// TwinCAT 3 PLC project RobotPlc
// ProgramVersion: 3.1.4024.0
// libraries:
//   Tc2_Standard, * (Beckhoff Automation GmbH)
//   Tc2_System, * (Beckhoff Automation GmbH)
//   Tc3_Module, * (Beckhoff Automation GmbH)
// project tree:
//   DUTs/ ST_FRUOPIn.TcDUT, ST_FRUOPOut.TcDUT, ST_FRConnection.TcDUT
//   / PlcTask.TcTTO
//   POUs/ FB_FRPower.TcPOU, FB_FRProgSelect.TcPOU, MAIN.TcPOU
// real-time tasks:
//   TASK PlcTask: cycle T#10ms, priority 20, ADS port 350
//   TASK EIP Scanner Task: cycle T#1ms, priority 1, ADS port 301
// I/O:
//   DEVICE Device 1 (TC3 EIP Scanner), AmsNetId 192.168.100.3.2.1
//     FANUC Robot R30iB+ // <INFO> 192.168.2.2, FANUC Robot R30iB+ (ProdCode: 4, Rev: 3.01, Mac: 8c:8c:aa:d6:16:77) </INFO> <EDS> C:\TwinCAT\3.1\Config\Io\EtherNetIP\FANUCROBOT_EIP_V900.EDS </EDS>
// variable links:
//   RobotPlc/RobotPlc Instance <-> Device 1 (TC3 EIP Scanner)/FANUC Robot R30iB+
//     PlcTask Inputs/MAIN.stFRConnection._EIPConnectionState <-> Inputs/State
//     PlcTask Inputs/MAIN.stFRConnection._rawIn <-> Connection 1 (Input/Output)/Inputs/noname0_arrBYTE[0]
//     PlcTask Inputs/MAIN.stFRConnection._rawIn @bit {8..56 step 8} <-> Connection 1 (Input/Output)/Inputs/noname0_arrBYTE[{1..7}]  (7 links)
//     PlcTask Outputs/MAIN.stFRConnection._rawOut <-> Connection 1 (Input/Output)/Outputs/noname0_arrBYTE[0]
//     PlcTask Outputs/MAIN.stFRConnection._rawOut @bit {8..56 step 8} <-> Connection 1 (Input/Output)/Outputs/noname0_arrBYTE[{1..7}]  (7 links)

CONFIGURATION RobotPlc
    RESOURCE PLC ON TwinCAT3
        TASK PlcTask(INTERVAL := T#10ms, PRIORITY := 20);
        PROGRAM MAIN WITH PlcTask : MAIN;
    END_RESOURCE
END_CONFIGURATION

// ---- DUTs/ST_FRUOPIn.TcDUT
TYPE ST_FRUOPIn :
STRUCT
	UI01_IMSTP : BIT;
	UI02_Hold : BIT;
	UI03_SFSPD : BIT;
	UI04_CycleStop : BIT;
	UI05_FaultReset : BIT;
	UI06_Start : BIT;
	UI07_Home : BIT;
	UI08_Enable : BIT;
	UI09_RSR1_PNS1 : BIT;
	UI10_RSR2_PNS2 : BIT;
	UI11_RSR3_PNS3 : BIT;
	UI12_RSR4_PNS4 : BIT;
	UI13_RSR5_PNS5 : BIT;
	UI14_RSR6_PNS6 : BIT;
	UI15_RSR7_PNS7 : BIT;
	UI16_RSR8_PNS8 : BIT;
	UI17_PNSStrobe : BIT;
	UI18_ProdStart : BIT;
	UI19,UI20,UI21,UI22
	,UI23,UI24,UI25,UI26
	,UI27,UI28,UI29,UI30
	,UI31,UI32 : BIT;
END_STRUCT
END_TYPE

// ---- DUTs/ST_FRUOPOut.TcDUT
TYPE ST_FRUOPOut :
STRUCT
	UO01_CmdEnabled : BIT;
	UO02_SystemReady : BIT;
	UO03_PrgRunning : BIT;
	UO04_PrgPaused : BIT;
	UO05_MotionHeld : BIT;
	UO06_Fault : BIT;
	UO07_AtPerch : BIT;
	UO08_TPEnabled : BIT;
	UO09_BattAlarm : BIT;
	UO10_Busy : BIT;
	UO11_ACK1_SNO1 : BIT;
	UO12_ACK2_SNO2 : BIT;
	UO13_ACK3_SNO3 : BIT;
	UO14_ACK4_SNO4 : BIT;
	UO15_ACK5_SNO5 : BIT;
	UO16_ACK6_SNO6 : BIT;
	UO17_ACK7_SNO7 : BIT;
	UO18_ACK8_SNO8 : BIT;
	UO19_SNACK : BIT;
	UO20_Reserved : BIT;
	UO21,UO22,UO23
	,UO24,UO25,UO26
	,UO27,UO28,UO29
	,UO30,UO31,UO32 : BIT;
END_STRUCT
END_TYPE

// ---- DUTs/ST_FRConnection.TcDUT
TYPE ST_FRConnection :
STRUCT
	_EIPConnectionState AT %I* : UINT;
	_rawIn AT %I*:ARRAY[0..7] OF BYTE;
	_rawOut AT %Q*:ARRAY[0..7] OF BYTE;
END_STRUCT
END_TYPE

// ---- POUs/MAIN.TcPOU
PROGRAM MAIN
VAR
	stFRConnection : ST_FRConnection;
	fbFRPower : FB_FRPower;
	fbFRProgSelect : FB_FRProgSelect;
	
	bIMSTP : BOOL;
	bHold : BOOL;
	bSFSPD : BOOL;
	bCycleStop : BOOL;
	bFaultReset : BOOL;
	bStart : BOOL;
	bHome : BOOL;
	bEnable : BOOL;

	bCmdEnabled : BOOL;
	bSystemReady : BOOL;
	bPrgRunning : BOOL;
	bPrgPaused : BOOL;
	bMotionHeld : BOOL;
	bFault : BOOL;
	bAtPerch : BOOL;
	bTPEnabled : BOOL;
	bBattAlarm : BOOL;
	bBusy : BOOL;
	
	bProgSelectExec : BOOL;
	bProgSelectDone : BOOL;
	bProgSelectBusy : BOOL;
	nProgSelectNo : USINT;
	nSelectedProgNo : USINT;
END_VAR

FRTest();

ACTION FRTest:
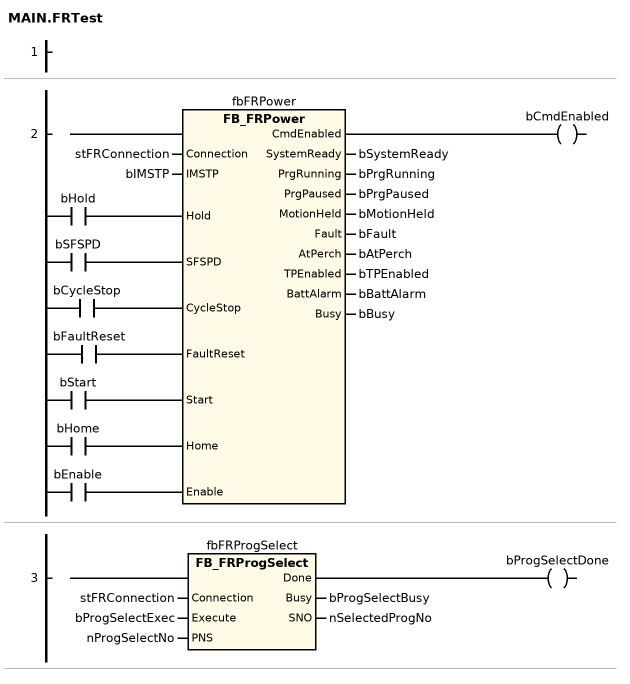
// NETWORK 1

// NETWORK 2
fbFRPower(
    Connection := stFRConnection,
    IMSTP := bIMSTP,
    Hold := bHold,
    SFSPD := bSFSPD,
    CycleStop := bCycleStop,
    FaultReset := bFaultReset,
    Start := bStart,
    Home := bHome,
    Enable := bEnable,
    SystemReady => bSystemReady,
    PrgRunning => bPrgRunning,
    PrgPaused => bPrgPaused,
    MotionHeld => bMotionHeld,
    Fault => bFault,
    AtPerch => bAtPerch,
    TPEnabled => bTPEnabled,
    BattAlarm => bBattAlarm,
    Busy => bBusy); // FB_FRPower
bCmdEnabled := fbFRPower.CmdEnabled;

// NETWORK 3
fbFRProgSelect(
    Connection := stFRConnection,
    Execute := bProgSelectExec,
    PNS := nProgSelectNo,
    Busy => bProgSelectBusy,
    SNO => nSelectedProgNo); // FB_FRProgSelect
bProgSelectDone := fbFRProgSelect.Done;
END_ACTION

END_PROGRAM

// ---- POUs/FB_FRPower.TcPOU
FUNCTION_BLOCK FB_FRPower
VAR_INPUT
	Connection : REFERENCE TO ST_FRConnection;
	IMSTP : BOOL;
	Hold : BOOL;
	SFSPD : BOOL;
	CycleStop : BOOL;
	FaultReset : BOOL;
	Start : BOOL;
	Home : BOOL;
	Enable : BOOL;
END_VAR
VAR_OUTPUT
	CmdEnabled : BOOL;
	SystemReady : BOOL;
	PrgRunning : BOOL;
	PrgPaused : BOOL;
	MotionHeld : BOOL;
	Fault : BOOL;
	AtPerch : BOOL;
	TPEnabled : BOOL;
	BattAlarm : BOOL;
	Busy : BOOL;
END_VAR
VAR
	stFRUOPIn : POINTER TO ST_FRUOPIn;
	stFRUOPOut : POINTER TO ST_FRUOPOut;
END_VAR

stFRUOPIn := ADR(Connection._rawOut);
stFRUOPOut := ADR(Connection._rawIn);

stFRUOPIn^.UI01_IMSTP := IMSTP;
stFRUOPIn^.UI02_Hold := Hold;
stFRUOPIn^.UI03_SFSPD := SFSPD;
stFRUOPIn^.UI04_CycleStop := CycleStop;
stFRUOPIn^.UI05_FaultReset := FaultReset;
stFRUOPIn^.UI06_Start := Start;
stFRUOPIn^.UI07_Home := Home;
stFRUOPIn^.UI08_Enable := Enable;

CmdEnabled := stFRUOPOut^.UO01_CmdEnabled;
SystemReady := stFRUOPOut^.UO02_SystemReady;
PrgRunning := stFRUOPOut^.UO03_PrgRunning;
PrgPaused := stFRUOPOut^.UO04_PrgPaused;
MotionHeld := stFRUOPOut^.UO05_MotionHeld;
Fault := stFRUOPOut^.UO06_Fault;
AtPerch := stFRUOPOut^.UO07_AtPerch;
TPEnabled := stFRUOPOut^.UO08_TPEnabled;
BattAlarm := stFRUOPOut^.UO09_BattAlarm;
Busy := stFRUOPOut^.UO09_BattAlarm;

END_FUNCTION_BLOCK

// ---- POUs/FB_FRProgSelect.TcPOU
FUNCTION_BLOCK FB_FRProgSelect
VAR_INPUT
	Connection : REFERENCE TO ST_FRConnection;
	Execute : BOOL;
	PNS : USINT;
END_VAR
VAR_OUTPUT
	Done : BOOL;
	Busy : BOOL;
	SNO : USINT;
END_VAR
VAR
	stFRUOPIn : POINTER TO ST_FRUOPIn;
	stFRUOPOut : POINTER TO ST_FRUOPOut;
	
	eProgState : (WAIT_EXEC, PNSSTROBE_TRIG, PNSSTROBE, WAIT_SNACK_DOWN, PROD_START);
	
	fbExecuteRTrig : R_TRIG;
	fbProdStartTON : TON := (PT := T#2S);
END_VAR

stFRUOPIn := ADR(Connection._rawOut);
stFRUOPOut := ADR(Connection._rawIn);

fbExecuteRTrig(CLK := Execute);

IF fbExecuteRTrig.Q AND eProgState = WAIT_EXEC THEN
	
	stFRUOPIn^.UI09_RSR1_PNS1 := PNS.0;
	stFRUOPIn^.UI10_RSR2_PNS2 := PNS.1;
	stFRUOPIn^.UI11_RSR3_PNS3 := PNS.2;
	stFRUOPIn^.UI12_RSR4_PNS4 := PNS.3;
	stFRUOPIn^.UI13_RSR5_PNS5 := PNS.4;
	stFRUOPIn^.UI14_RSR6_PNS6 := PNS.5;
	stFRUOPIn^.UI15_RSR7_PNS7 := PNS.6;
	stFRUOPIn^.UI16_RSR8_PNS8 := PNS.7;
	
	eProgState := PNSSTROBE;
END_IF

CASE eProgState OF
	WAIT_EXEC:
		// Wait for Execute raising edge.
	PNSSTROBE:
		Done := FALSE;
		Busy := TRUE;
		stFRUOPIn^.UI17_PNSStrobe := TRUE;
		
		IF stFRUOPOut^.UO19_SNACK THEN

			SNO.0 := stFRUOPOut^.UO11_ACK1_SNO1;
			SNO.1 := stFRUOPOut^.UO12_ACK2_SNO2;
			SNO.2 := stFRUOPOut^.UO13_ACK3_SNO3;
			SNO.3 := stFRUOPOut^.UO14_ACK4_SNO4;
			SNO.4 := stFRUOPOut^.UO15_ACK5_SNO5;
			SNO.5 := stFRUOPOut^.UO16_ACK6_SNO6;
			SNO.6 := stFRUOPOut^.UO17_ACK7_SNO7;
			SNO.7 := stFRUOPOut^.UO18_ACK8_SNO8;

			eProgState := WAIT_SNACK_DOWN;
		END_IF
		
	WAIT_SNACK_DOWN:
		IF NOT stFRUOPOut^.UO19_SNACK THEN
			eProgState := PROD_START;
		END_IF
	PROD_START:
		stFRUOPIn^.UI18_ProdStart := TRUE;
		fbProdStartTON(IN := TRUE);
		
		IF fbProdStartTON.Q OR stFRUOPOut^.UO03_PrgRunning THEN
			stFRUOPIn^.UI17_PNSStrobe := FALSE;
			stFRUOPIn^.UI18_ProdStart := FALSE;
			fbProdStartTON(IN := FALSE);
			Done := TRUE;
			Busy := FALSE;
			eProgState := WAIT_EXEC;
		END_IF
		
END_CASE

END_FUNCTION_BLOCK
